// TIA Portal V17 export
// export: Created 2022-07-28T18:02:46.6658222Z, ExportSetting None, DisplayName Totally Integrated Automation Portal, DisplayVersion V17, DisplayName TIA Portal Openness, DisplayVersion V17, DisplayName TIA Portal Teamcenter Gateway, DisplayVersion V17, DisplayName TIA Portal Version Control Interface, DisplayVersion V17, DisplayName TIA Portal Test Suite Advanced, DisplayVersion V17, DisplayName SINAMICS Startdrive Advanced, DisplayVersion V17, DisplayName SINAMICS DCC, DisplayVersion V17, DisplayName SINAMICS Startdrive G130, G150, S120, S150, SINAMICS MV, S210, DisplayVersion V17, DisplayName SINAMICS Startdrive G110M, G120, G120C, G120D, G120P, G115D, DisplayVersion V17, DisplayName STEP 7 Professional, DisplayVersion V17, DisplayName SIMATIC Energy Suite, DisplayVersion V17, DisplayName STEP 7 CFC, DisplayVersion V17, DisplayName STEP 7 Safety, DisplayVersion V17, DisplayName WinCC Advanced / Unified PC, DisplayVersion V17, DisplayName SIMATIC Visualization Architect, DisplayVersion V17
FUNCTION "Begin_FC" : Void   // FC1, SCL
{ S7_Optimized_Access := 'TRUE' }
// stored: SetENOAutomatically false
   VAR_TEMP
      twErrRetVal : Int;
      i : Int;
      j : Int;
      Zero_CycleInfo : "Lib_PLC_CycleInfo";
      arr_CycleInfo : Array[0..9, 0..15] of "Lib_PLC_CycleInfo";
      Zero : Struct
         "B" : Byte;
         W : Word;
         D : DWord;
      END_STRUCT;
      Bufer : Struct
         "B" : Byte;
         W : Word;
         D : DWord;
      END_STRUCT;
      tmp_State : Byte;
      tmp_Alarm : DWord;
      tmp_State_j : Byte;
      tmp_Alarm_j : DWord;
      Max_Number_Groups : Int;
      Max_Number_ButtonInGroup : Int;
   END_VAR
BEGIN
   //Number of objects in Plant
   "D_General_ProgramDATA".ui_MaxObjects := 30;

   //------------------------------
   REGION CycleInfo
       //Збір і обробка інформації від груп обєктів про стани та аварії протягом циклу та передача на HMI 
       REGION завантаження в перевірка розмірк масиву Груп/рідгруп для CycleInfo
           #Max_Number_Groups := "D_PLC_CycleInfo_DATA".Config.Max_Number_Groups;
           #Max_Number_ButtonInGroup := "D_PLC_CycleInfo_DATA".Config.Max_Number_ButtonInGroup;
           IF #Max_Number_Groups > 9 THEN
               "D_PLC_CycleInfo_DATA".Config.Max_Number_Groups := 9;
           END_IF;
           IF #Max_Number_ButtonInGroup > 15 THEN
               "D_PLC_CycleInfo_DATA".Config.Max_Number_ButtonInGroup := 15;
           END_IF;
           IF #Max_Number_Groups < 1 THEN
               "D_PLC_CycleInfo_DATA".Config.Max_Number_Groups := 1;
           END_IF;
           IF #Max_Number_ButtonInGroup < 1 THEN
               "D_PLC_CycleInfo_DATA".Config.Max_Number_ButtonInGroup := 1;
           END_IF;
       END_REGION

       REGION обробка даних від Obj
           // i - Групи, i = 0 - обєдані дані груп  i=1..9
           // j - підгрупи, j = 0 - обєдані дані підгруп j=1..15 групи i
           //---------------------------------------
           // завантаження в #arr_CycleInfo CMD_GLOBAL від HMI для всіх груп і підгруп #i >= 0 AND #j >= 0)
           // завантаження в #arr_CycleInfo даних зібраних від Obj для усіх  підгруп (#i > 0 AND #j > 0)
           FOR #i := 0 TO #Max_Number_Groups DO
               FOR #j := 0 TO #Max_Number_ButtonInGroup DO // Statement section FOR
                   IF #i > 0 AND #j > 0 THEN
                       #arr_CycleInfo[#i, #j] := "D_PLC_CycleInfo_DATA".Grp_Obj[#i, #j];
                   END_IF;
                   #arr_CycleInfo[#i, #j].CMD_GLOBAL := "D_PLC_CycleInfo_DATA"."Grp_HMI&CNTR"[#i, #j].CMD_GLOBAL;
                   //"D_PLC_CycleInfo_DATA"."Grp_HMI&CNTR"[#i, #j].CMD_GLOBAL := 0;
                   //#arr_CycleInfo[#i, #j].CMD_GLOBAL_SP := "D_PLC_CycleInfo_DATA"."Grp_HMI&CNTR"[#i, #j].CMD_GLOBAL_SP;
                   //#arr_CycleInfo[#i, #j].CMD_GLOBAL := 0;
               END_FOR;
           END_FOR;

           FOR #i := 1 TO #Max_Number_Groups DO
               #tmp_Alarm_j := 0;
               #tmp_State_j := 0;
               //--------------
               // обробка CMD_GLOBAL групи i
               IF #arr_CycleInfo[0, 0].CMD_GLOBAL <> 0 THEN
                   #arr_CycleInfo[#i, 0].CMD_GLOBAL := #arr_CycleInfo[0, 0].CMD_GLOBAL;
                   "D_PLC_CycleInfo_DATA"."Grp_HMI&CNTR"[#i, 0].CMD_GLOBAL := #arr_CycleInfo[0, 0].CMD_GLOBAL;
               END_IF;
               // --------------
               FOR #j := 1 TO #Max_Number_ButtonInGroup DO // Statement section FOR
                   // обробка лічильиків підгрупи j та Формування загального лічильика групи i
                   #arr_CycleInfo[#i, 0].Counter.Alarm := #arr_CycleInfo[#i, 0].Counter.Alarm + #arr_CycleInfo[#i, #j].Counter.Alarm;
                   #arr_CycleInfo[#i, 0].Counter.Warning := #arr_CycleInfo[#i, 0].Counter.Warning + #arr_CycleInfo[#i, #j].Counter.Warning;
                   #arr_CycleInfo[#i, 0].Counter.ErrorBad := #arr_CycleInfo[#i, 0].Counter.ErrorBad + #arr_CycleInfo[#i, #j].Counter.ErrorBad;
                   #arr_CycleInfo[#i, 0].Counter.Forced := #arr_CycleInfo[#i, 0].Counter.Forced + #arr_CycleInfo[#i, #j].Counter.Forced;
                   #arr_CycleInfo[#i, 0].Counter.Manual := #arr_CycleInfo[#i, 0].Counter.Manual + #arr_CycleInfo[#i, #j].Counter.Manual;
                   #arr_CycleInfo[#i, 0].Counter.Interlocked := #arr_CycleInfo[#i, 0].Counter.Interlocked + #arr_CycleInfo[#i, #j].Counter.Interlocked;
                   #arr_CycleInfo[#i, 0].Counter.Simulation := #arr_CycleInfo[#i, 0].Counter.Simulation + #arr_CycleInfo[#i, #j].Counter.Simulation;
                   //--------------
                   // обробка Alarm підгрупи j
                   GATHER(IN := #arr_CycleInfo[#i, #j].Alarm,
                          OUT => #Bufer.D);
                   #tmp_Alarm_j := #tmp_Alarm_j OR #Bufer.D;
                   // STW підгрупи j  та Формування загального STW групи i
                   #arr_CycleInfo[#i, #j].STW := #Bufer.D;
                   //--------------
                   // обробка State підгрупи j
                   GATHER(IN := #arr_CycleInfo[#i, #j].State,
                          OUT => #Bufer.B);
                   #tmp_State_j := #tmp_State_j OR #Bufer.B;
                   // STW підгрупи j  та Формування загального STW групи i
                   #arr_CycleInfo[#i, #j].STW.%B3 := #Bufer.B;
                   //--------------
                   // обробка CMD_GLOBAL підгрупи j
                   IF #arr_CycleInfo[#i, 0].CMD_GLOBAL <> 0 THEN
                       #arr_CycleInfo[#i, #j].CMD_GLOBAL := #arr_CycleInfo[#i, 0].CMD_GLOBAL;
                       "D_PLC_CycleInfo_DATA"."Grp_HMI&CNTR"[#i, #j].CMD_GLOBAL := #arr_CycleInfo[#i, 0].CMD_GLOBAL;
                   END_IF;
                   //_#arr_CycleInfo[#i, #j].CMD_GLOBAL := #arr_CycleInfo[#i, #j].CMD_GLOBAL_SP;
                   //_#arr_CycleInfo[#i, #j].CMD_GLOBAL_SP := 0;

               END_FOR;
               //--------------
               // Формування загального Alarm групи i
               SCATTER(IN := #tmp_Alarm_j,
                       OUT => #arr_CycleInfo[#i, 0].Alarm);
               // Формування загального State групи i
               SCATTER(IN := #tmp_State_j,
                       OUT => #arr_CycleInfo[#i, 0].State);
               // Формування загального STW групи i
               #arr_CycleInfo[#i, 0].STW := #tmp_Alarm_j;
               #arr_CycleInfo[#i, 0].STW.%B3 := #tmp_State_j;
               //--------------
               // обробка лічильиків групи i т Формування загального лічильика системи (#i = 0 AND #j = 0)
               #arr_CycleInfo[0, 0].Counter.Alarm := #arr_CycleInfo[0, 0].Counter.Alarm + #arr_CycleInfo[#i, 0].Counter.Alarm;
               #arr_CycleInfo[0, 0].Counter.Warning := #arr_CycleInfo[0, 0].Counter.Warning + #arr_CycleInfo[#i, 0].Counter.Warning;
               #arr_CycleInfo[0, 0].Counter.ErrorBad := #arr_CycleInfo[0, 0].Counter.ErrorBad + #arr_CycleInfo[#i, 0].Counter.ErrorBad;
               #arr_CycleInfo[0, 0].Counter.Forced := #arr_CycleInfo[0, 0].Counter.Forced + #arr_CycleInfo[#i, 0].Counter.Forced;
               #arr_CycleInfo[0, 0].Counter.Manual := #arr_CycleInfo[0, 0].Counter.Manual + #arr_CycleInfo[#i, 0].Counter.Manual;
               #arr_CycleInfo[0, 0].Counter.Interlocked := #arr_CycleInfo[0, 0].Counter.Interlocked + #arr_CycleInfo[#i, 0].Counter.Interlocked;
               #arr_CycleInfo[0, 0].Counter.Simulation := #arr_CycleInfo[0, 0].Counter.Simulation + #arr_CycleInfo[#i, 0].Counter.Simulation;
               //#arr_CycleInfo[#i, 0].Counter := #Zero_CycleInfo.Counter;
               //--------------
               // обробка Alarm групи i
               GATHER(IN := #arr_CycleInfo[#i, 0].Alarm,
                      OUT => #Bufer.D);
               #tmp_Alarm := #tmp_Alarm OR #Bufer.D;
               // #arr_CycleInfo[#i, 0].Alarm := #Zero_CycleInfo.Alarm;
               //--------------
               // обробка State групи i
               GATHER(IN := #arr_CycleInfo[#i, 0].State,
                      OUT => #Bufer.B);
               #tmp_State := #tmp_State OR #Bufer.B;
               //#arr_CycleInfo[#i, 0].State := #Zero_CycleInfo.State;


           END_FOR;


           //--------------
           // Формування загального Alarm системи (#i = 0 AND #j = 0)
           SCATTER(IN := #tmp_Alarm,
                   OUT => #arr_CycleInfo[0, 0].Alarm);
           // Формування загального State системи (#i = 0 AND #j = 0)
           SCATTER(IN := #tmp_State,
                   OUT => #arr_CycleInfo[0, 0].State);
           // Формування загального STW системи (#i = 0 AND #j = 0)
           #arr_CycleInfo[0, 0].STW := #tmp_Alarm;
           #arr_CycleInfo[0, 0].STW.%B3 := #tmp_State;
           //----------------------------------------------------------------------------------------------------------------

       END_REGION
       //----------------------------------------------------------------------------------------------------------------
       // Дані системи (#i = 0 AND #j = 0) --> "1_PLC_DATA".CycleInfo 
       "D_PLC".CycleInfo := #arr_CycleInfo[0, 0];
       // Всі Дані --> HMI
       "D_PLC_CycleInfo_DATA"."Grp_HMI&CNTR" := #arr_CycleInfo;
       //----------------------------------------------------------------------------------------------------------------
       //Ініціалізація нового циклу для Obj / скидання даних / передача команд від  HMI -->Obj
       FOR #i := 0 TO #Max_Number_Groups DO
           FOR #j := 0 TO #Max_Number_ButtonInGroup DO // Statement section FOR
               #arr_CycleInfo[#i, #j] := #Zero_CycleInfo;
               #arr_CycleInfo[#i, #j].CMD_GLOBAL := "D_PLC_CycleInfo_DATA"."Grp_HMI&CNTR"[#i, #j].CMD_GLOBAL;
               "D_PLC_CycleInfo_DATA"."Grp_HMI&CNTR"[#i, #j].CMD_GLOBAL := 0;

           END_FOR;
       END_FOR;

       "D_PLC_CycleInfo_DATA".Grp_Obj := #arr_CycleInfo;


   END_REGION

   REGION General bits
       //Read data from HMI
       IF "D_General_HMI".i_CMD <> 0
       THEN
           "D_General_ProgramDATA".i_CMD := "D_General_HMI".i_CMD;
           "D_General_HMI".i_CMD := 0;
       END_IF;

       //General bits 
       "D_General_ProgramDATA".RestartPLC := "FirstScan";

       CASE "D_General_ProgramDATA".i_CMD OF
           1000:  //ES from HMI
               "D_General_ProgramDATA".ES_HMI_Global := false;
           1001:  //Global reset
               "D_General_ProgramDATA".ResetGlobal := true;
           ELSE  
               ;
       END_CASE;

       IF "D_General_ProgramDATA".ResetGlobal
       THEN
           "D_General_ProgramDATA".ES_HMI_Global := true;
       END_IF;

       "D_General_ProgramDATA".ES_Fld_Global := "Internal_H05_FB_DB".Q_KM_SafRelay_Ok;
   END_REGION

   REGION Proccess internal signals (fuses, safety, ect)
       "Internal_H01_FB_DB"(I_CmdGeneralReset:="D_General_ProgramDATA".ResetGlobal,
                            IR_CycleTime:="D_PLC".TIME_TCK.cyclic_sec_R,
                            I_Initialization:="D_General_ProgramDATA".RestartPLC,
                            I_One_1s:="D_PLC".PLS.P1S,
                            I_KV_Ok := "I_PRE_H01_001_KV1_PSL400" ,
                            I_QF_Trans_Ok := "I_PRE_H01_003_Q1_PSL230" ,
                            I_QF_Oper230_Ok := "I_PRE_H01_003_F1_PSL230" ,
                            I_QF_Oper24_Ok := "I_PRE_H01_003_F2_PSL230" ,
                            I_QF_Saf_Ok := "I_PRE_H01_003_F3_PSL230" ,
                            I_QF_KM_Ok := "I_PRE_H01_003_F4_PSL230" ,
                            I_QF_Gas_Ok := "I_PRE_H01_003_F5_PSL230" ,
                            I_QF_VlvSaf_Ok := "I_PRE_H01_003_F6_PSL230" ,
                            I_QF_Spare_Ok := "I_PRE_H01_003_F7_PSL230",
                            QW_STW=>"Internal_H01_FB_DB".QW_STW,
                            Q_Reset=>"Internal_H01_FB_DB".Q_Reset,
                            Q_SomeErr=>"Internal_H01_FB_DB".Q_SomeErr,
                            Q_KV_Ok=>"Internal_H01_FB_DB".Q_KV_Ok,
                            Q_QF_Trans_Ok=>"Internal_H01_FB_DB".Q_QF_Trans_Ok,
                            Q_QF_Oper230_Ok=>"Internal_H01_FB_DB".Q_QF_Oper230_Ok,
                            Q_QF_Oper24_Ok=>"Internal_H01_FB_DB".Q_QF_Oper24_Ok,
                            Q_QF_Saf_Ok=>"Internal_H01_FB_DB".Q_QF_Saf_Ok,
                            Q_QF_KM_Ok=>"Internal_H01_FB_DB".Q_QF_KM_Ok,
                            Q_QF_Gas_Ok=>"Internal_H01_FB_DB".Q_QF_Gas_Ok,
                            Q_QF_VlvSaf_Ok=>"Internal_H01_FB_DB".Q_QF_VlvSaf_Ok,
                            Q_QF_Spare_Ok=>"Internal_H01_FB_DB".Q_QF_Spare_Ok );

       "Internal_H05_FB_DB"(I_CmdGeneralReset:="D_General_ProgramDATA".ResetGlobal,
                            IR_CycleTime:="D_PLC".TIME_TCK.cyclic_sec_R,
                            I_Initialization:="D_General_ProgramDATA".RestartPLC,
                            I_One_1s:="D_PLC".PLS.P1S,
                            I_Sup24_Ok := "I_PRE_H05_004_T1_PSL24" ,
                            I_UPS_Alarm_Ok := NOT "I_PRE_H05_004_K1_1_PSL24" ,
                            I_UPS_Bat_Ok := NOT "I_PRE_H05_004_K1_2_PSL24" ,
                            I_QF_DQ_Ok := "I_PRE_H05_004_F4_PSL24" ,
                            I_QF_AI_Ok := "I_PRE_H05_004_F5_PSL24" ,
                            I_QF_AQ_Ok := "I_PRE_H05_004_F6_PSL24" ,
                            I_QF_Desmet_IM_Ok := "I_PRE_H05_004_F7_PSL24" ,
                            I_QF_Desmet_DI_DQ_Ok := "I_PRE_H05_004_F8_PSL24" ,
                            I_QF_Desmet_AI_AQ_Ok := "I_PRE_H05_004_F9_PSL24" ,
                            I_QF_Inv_Ctrl_Ok := "I_PRE_H05_004_F10_PSL24" ,
                            I_QF_Inv_STO_Ok := "I_PRE_H05_004_F11_PSL24" ,
                            I_QF_Internal_Ok := "I_PRE_H05_004_F12_PSL24" ,
                            I_QF_SafRelay_Ok := "I_PRE_H05_004_F13_PSL24" ,
                            I_QF_Analog_Ok := "I_PRE_H05_004_F14_PSL24" ,
                            I_QF_ThermoRelay_Ok := "I_PRE_H05_004_F15_PSL24" ,
                            I_QF_VlvDisFoam_Ok := "I_PRE_H05_004_F16_PSL24" ,
                            I_QF_FlowMeters_Ok := "I_PRE_H05_004_F17_PSL24" ,
                            I_QF_VlvVitamin_Ok := "I_PRE_H05_004_F18_PSL24" ,
                            I_QF_DI_DQ_1_Ok := "I_PRE_H05_004_F19_PSL24" ,
                            I_QF_DI_DQ_2_Ok := "I_PRE_H05_004_F20_PSL24" ,
                            I_QS_Scalance_Ok := "I_PRE_H05_004_F21_PSL24" ,
                            I_SB_ES_Box_Ok := "I_PRE_H05_005_SB1_SAF" ,
                            I_SB_ES_Ack_Ok := "I_PRE_H05_005_SB2_SAF" ,
                            I_KM_SafRelay_Ok := "I_PRE_H05_005_KM2_SAF" ,
                            QW_STW=>"Internal_H05_FB_DB".QW_STW,
                            QW_MW1=>"Internal_H05_FB_DB".QW_MW1,
                            QW_MW2=>"Internal_H05_FB_DB".QW_MW2,
                            QW_MW3=>"Internal_H05_FB_DB".QW_MW3,
                            Q_Reset=> "Q_PRE_H05_005_KL1_SAF",
                            Q_SomeErr=>"Internal_H05_FB_DB".Q_SomeErr,
                            Q_Sup24_Ok=>"Internal_H05_FB_DB".Q_Sup24_Ok,
                            Q_UPS_Alarm_Ok=>"Internal_H05_FB_DB".Q_UPS_Alarm_Ok,
                            Q_UPS_Bat_Ok=>"Internal_H05_FB_DB".Q_UPS_Bat_Ok,
                            Q_QF_DQ_Ok=>"Internal_H05_FB_DB".Q_QF_DQ_Ok,
                            Q_QF_AI_Ok=>"Internal_H05_FB_DB".Q_QF_AI_Ok,
                            Q_QF_AQ_Ok=>"Internal_H05_FB_DB".Q_QF_AQ_Ok,
                            Q_QF_Desmet_IM_Ok=>"Internal_H05_FB_DB".Q_QF_Desmet_IM_Ok,
                            Q_QF_Desmet_DI_DQ_Ok=>"Internal_H05_FB_DB".Q_QF_Desmet_DI_DQ_Ok,
                            Q_QF_Desmet_AI_AQ_Ok=>"Internal_H05_FB_DB".Q_QF_Desmet_AI_AQ_Ok,
                            Q_QF_Inv_Ctrl_Ok=>"Internal_H05_FB_DB".Q_QF_Inv_Ctrl_Ok,
                            Q_QF_Inv_STO_Ok=>"Internal_H05_FB_DB".Q_QF_Inv_STO_Ok,
                            Q_QF_Internal_Ok=>"Internal_H05_FB_DB".Q_QF_Internal_Ok,
                            Q_QF_SafRelay_Ok=>"Internal_H05_FB_DB".Q_QF_SafRelay_Ok,
                            Q_QF_Analog_Ok=>"Internal_H05_FB_DB".Q_QF_Analog_Ok,
                            Q_QF_ThermoRelay_Ok=>"Internal_H05_FB_DB".Q_QF_ThermoRelay_Ok,
                            Q_QF_VlvDisFoam_Ok=>"Internal_H05_FB_DB".Q_QF_VlvDisFoam_Ok,
                            Q_QF_FlowMeters_Ok=>"Internal_H05_FB_DB".Q_QF_FlowMeters_Ok,
                            Q_QF_VlvVitamin_Ok=>"Internal_H05_FB_DB".Q_QF_VlvVitamin_Ok,
                            Q_QF_DI_DQ_1_Ok=>"Internal_H05_FB_DB".Q_QF_DI_DQ_1_Ok,
                            Q_QF_DI_DQ_2_Ok=>"Internal_H05_FB_DB".Q_QF_DI_DQ_2_Ok,
                            Q_QS_Scalance_Ok=>"Internal_H05_FB_DB".Q_QS_Scalance_Ok,
                            Q_KM_SafRelay_Ok=>"Internal_H05_FB_DB".Q_KM_SafRelay_Ok);

       "Q_PRE_H05_005_SB2_SAF" := NOT  "Internal_H05_FB_DB".Q_KM_SafRelay_Ok
       AND "Clock_1Hz";
   END_REGION

   REGION Proccess IO devices states
       "D_PN_IO_Status".i_RetVal  := DeviceStates(LADDR := "D_PN_IO_Status".hw_LADDR,
                                                  MODE := "D_PN_IO_Status".ui_Mode,
                                                  STATE := "D_PN_IO_Status".States);

       //Proccess states with reset
       FOR #j := 0 TO 1023 DO
           IF "D_PN_IO_Status".States[#j]
           THEN
               "D_PN_IO_Status".States_Proc[#j] := true;
           END_IF;

           IF (NOT "D_PN_IO_Status".States[#j]
               AND "D_General_ProgramDATA".ResetGlobal)
               OR "D_General_ProgramDATA".RestartPLC
           THEN
               "D_PN_IO_Status".States_Proc[#j] := false;
           END_IF;
       END_FOR;

   END_REGION

   REGION Wrap general states into words to HMI

       //Some safety fault is active
       "D_General_HMI".w_MW1.%X0 := NOT "Internal_H05_FB_DB".Q_KM_SafRelay_Ok
       OR NOT "Internal_H05_FB_DB".Q_QF_SafRelay_Ok
       OR NOT "Internal_H05_FB_DB".Q_QF_Internal_Ok
       OR NOT "Internal_H01_FB_DB".I_QF_Gas_Ok
       OR NOT "Internal_H01_FB_DB".I_QF_VlvSaf_Ok
       OR "D_InOut".XV6_Safe.Cmd_Open
       OR NOT "D_InOut".DI7_S1.DescreteValue
       OR NOT "D_InOut".DI7_S3.DescreteValue
       OR NOT "D_General_ProgramDATA".ES_HMI_Global;

       //Some fault with IO devices is active
       "D_General_HMI".w_MW1.%X1 := "D_PN_IO_Status".States_Proc[0];

       //Some faults in H01
       "D_General_HMI".w_MW1.%X2 := "Internal_H01_FB_DB".Q_SomeErr;

       //Some faults in H05
       "D_General_HMI".w_MW1.%X3 := "Internal_H05_FB_DB".Q_SomeErr;

       //General bits
       REGION Word #MW2 - safety units
           "D_General_HMI".w_MW2.%X0 := "D_InOut".XV6_Safe.Cmd_Open; //Command to safe valve for close
           "D_General_HMI".w_MW2.%X1 := NOT "D_InOut".DI7_S1.DescreteValue;  //Gas sensor - H level (Horn)
           "D_General_HMI".w_MW2.%X2 := NOT "D_InOut".DI7_S3.DescreteValue;  //Gas sensor - HH level (Close safety valve XV6)
           "D_General_HMI".w_MW2.%X3 := NOT "Internal_H05_FB_DB".Q_KM_SafRelay_Ok; //KM of Safety relay don't switched on
           "D_General_HMI".w_MW2.%X4 := NOT "Internal_H05_FB_DB".Q_QF_SafRelay_Ok; //QF of Safety relay don't switched on
           "D_General_HMI".w_MW2.%X5 := NOT "Internal_H01_FB_DB".I_QF_Gas_Ok; //QF of Gas sensor don't switched on
           "D_General_HMI".w_MW2.%X6 := NOT "Internal_H01_FB_DB".I_QF_VlvSaf_Ok; //QF of Safety valve don't switched on
           "D_General_HMI".w_MW2.%X7 := NOT "I_PRE_H05_005_SB1_SAF"; //Emergency stop push button on the door of box H05 was pressed
           "D_General_HMI".w_MW2.%X8 := NOT "D_General_ProgramDATA".ES_HMI_Global; //Emergency stop from HMI
           "D_General_HMI".w_MW2.%X9 := false;
           "D_General_HMI".w_MW2.%X10 := false;
           "D_General_HMI".w_MW2.%X11 := false;
           "D_General_HMI".w_MW2.%X12 := false;
           "D_General_HMI".w_MW2.%X13 := false;
           "D_General_HMI".w_MW2.%X14 := false;

       END_REGION

       REGION Word #MW3 - connections with IO devices
           "D_General_HMI".w_MW3.%X0 := "D_PN_IO_Status".States_Proc[1];  //H2UZ1
           "D_General_HMI".w_MW3.%X1 := "D_PN_IO_Status".States_Proc[2];  //H3UZ1
           "D_General_HMI".w_MW3.%X2 := "D_PN_IO_Status".States_Proc[3];  //H4UZ1
           "D_General_HMI".w_MW3.%X3 := "D_PN_IO_Status".States_Proc[4];  //BoilUZ1
           "D_General_HMI".w_MW3.%X4 := false;
           "D_General_HMI".w_MW3.%X5 := false;
           "D_General_HMI".w_MW3.%X6 := false;
           "D_General_HMI".w_MW3.%X7 := false;
           "D_General_HMI".w_MW3.%X8 := false;
           "D_General_HMI".w_MW3.%X9 := false;
           "D_General_HMI".w_MW3.%X10 := false;
           "D_General_HMI".w_MW3.%X11 := false;
           "D_General_HMI".w_MW3.%X12 := false;
           "D_General_HMI".w_MW3.%X13 := false;
           "D_General_HMI".w_MW3.%X14 := false;

       END_REGION

       REGION Word #MW4
           "D_General_HMI".w_MW4.%X0 := false;
           "D_General_HMI".w_MW4.%X1 := false;
           "D_General_HMI".w_MW4.%X2 := false;
           "D_General_HMI".w_MW4.%X3 := false;
           "D_General_HMI".w_MW4.%X4 := false;
           "D_General_HMI".w_MW4.%X5 := false;
           "D_General_HMI".w_MW4.%X6 := false;
           "D_General_HMI".w_MW4.%X7 := false;
           "D_General_HMI".w_MW4.%X8 := false;
           "D_General_HMI".w_MW4.%X9 := false;
           "D_General_HMI".w_MW4.%X10 := false;
           "D_General_HMI".w_MW4.%X11 := false;
           "D_General_HMI".w_MW4.%X12 := false;
           "D_General_HMI".w_MW4.%X13 := false;
           "D_General_HMI".w_MW4.%X14 := false;

       END_REGION

       REGION Word #MW5
           "D_General_HMI".w_MW5.%X0 := false;
           "D_General_HMI".w_MW5.%X1 := false;
           "D_General_HMI".w_MW5.%X2 := false;
           "D_General_HMI".w_MW5.%X3 := false;
           "D_General_HMI".w_MW5.%X4 := false;
           "D_General_HMI".w_MW5.%X5 := false;
           "D_General_HMI".w_MW5.%X6 := false;
           "D_General_HMI".w_MW5.%X7 := false;
           "D_General_HMI".w_MW5.%X8 := false;
           "D_General_HMI".w_MW5.%X9 := false;
           "D_General_HMI".w_MW5.%X10 := false;
           "D_General_HMI".w_MW5.%X11 := false;
           "D_General_HMI".w_MW5.%X12 := false;
           "D_General_HMI".w_MW5.%X13 := false;
           "D_General_HMI".w_MW5.%X14 := false;

       END_REGION

       REGION Word #MW6
           "D_General_HMI".w_MW6.%X0 := false;
           "D_General_HMI".w_MW6.%X1 := false;
           "D_General_HMI".w_MW6.%X2 := false;
           "D_General_HMI".w_MW6.%X3 := false;
           "D_General_HMI".w_MW6.%X4 := false;
           "D_General_HMI".w_MW6.%X5 := false;
           "D_General_HMI".w_MW6.%X6 := false;
           "D_General_HMI".w_MW6.%X7 := false;
           "D_General_HMI".w_MW6.%X8 := false;
           "D_General_HMI".w_MW6.%X9 := false;
           "D_General_HMI".w_MW6.%X10 := false;
           "D_General_HMI".w_MW6.%X11 := false;
           "D_General_HMI".w_MW6.%X12 := false;
           "D_General_HMI".w_MW6.%X13 := false;
           "D_General_HMI".w_MW6.%X14 := false;

       END_REGION

       REGION Word #MW8
           "D_General_HMI".w_MW8.%X0 := false;
           "D_General_HMI".w_MW8.%X1 := false;
           "D_General_HMI".w_MW8.%X2 := false;
           "D_General_HMI".w_MW8.%X3 := false;
           "D_General_HMI".w_MW8.%X4 := false;
           "D_General_HMI".w_MW8.%X5 := false;
           "D_General_HMI".w_MW8.%X6 := false;
           "D_General_HMI".w_MW8.%X7 := false;
           "D_General_HMI".w_MW8.%X8 := false;
           "D_General_HMI".w_MW8.%X9 := false;
           "D_General_HMI".w_MW8.%X10 := false;
           "D_General_HMI".w_MW8.%X11 := false;
           "D_General_HMI".w_MW8.%X12 := false;
           "D_General_HMI".w_MW8.%X13 := false;
           "D_General_HMI".w_MW8.%X14 := false;

       END_REGION

       REGION Word #MW9
           "D_General_HMI".w_MW9.%X0 := false;
           "D_General_HMI".w_MW9.%X1 := false;
           "D_General_HMI".w_MW9.%X2 := false;
           "D_General_HMI".w_MW9.%X3 := false;
           "D_General_HMI".w_MW9.%X4 := false;
           "D_General_HMI".w_MW9.%X5 := false;
           "D_General_HMI".w_MW9.%X6 := false;
           "D_General_HMI".w_MW9.%X7 := false;
           "D_General_HMI".w_MW9.%X8 := false;
           "D_General_HMI".w_MW9.%X9 := false;
           "D_General_HMI".w_MW9.%X10 := false;
           "D_General_HMI".w_MW9.%X11 := false;
           "D_General_HMI".w_MW9.%X12 := false;
           "D_General_HMI".w_MW9.%X13 := false;
           "D_General_HMI".w_MW9.%X14 := false;

       END_REGION

       REGION Word #MW10
           "D_General_HMI".w_MW10.%X0 := false;
           "D_General_HMI".w_MW10.%X1 := false;
           "D_General_HMI".w_MW10.%X2 := false;
           "D_General_HMI".w_MW10.%X3 := false;
           "D_General_HMI".w_MW10.%X4 := false;
           "D_General_HMI".w_MW10.%X5 := false;
           "D_General_HMI".w_MW10.%X6 := false;
           "D_General_HMI".w_MW10.%X7 := false;
           "D_General_HMI".w_MW10.%X8 := false;
           "D_General_HMI".w_MW10.%X9 := false;
           "D_General_HMI".w_MW10.%X10 := false;
           "D_General_HMI".w_MW10.%X11 := false;
           "D_General_HMI".w_MW10.%X12 := false;
           "D_General_HMI".w_MW10.%X13 := false;
           "D_General_HMI".w_MW10.%X14 := false;

       END_REGION


   END_REGION


   "1_PLC_FB_DB"();
   "Inputs_FC"();
END_FUNCTION
